# EPICS SNL sequencer program: test/validate/assign.st
program assign_test

%%#include <stdlib.h>
%%#include "epicsUnitTest.h"

int x = 0;
assign x;

foreign pvStatERROR;

#define NTESTS 3

entry {
    testPlan(NTESTS);
}

ss w {
    int n = 1;
    state w {
        when(n > NTESTS) {
        } exit
        when (delay(0.01)) {
            int status;
            x = !x;
            status = pvPut(x);
            testOk1(status==pvStatERROR);
            n++;
        } state w
    }
}

ss r {
    state yes {
        when (!x) {
        } state no
    }
    state no {
        when (x) {
        } state yes
    }
}

exit {
    testDone();
    exit(0);
}
